(* IEC 61131-3 sources: ATCMcontrol_Engineering/src/TargetBase/Libs/ATCM_File, 19 files *)

(* ---- F_ERROR_STRING.st ---- *)
(*[[
    UserURL= "ATCMfile:F_ERROR_STRING.htm"
]]*)

(* F_ERROR_STRING
 * ----------------------------------------------------------------------------
 * Retrieves the error text that corresponds to the error number.
 *
 * in   ERRCD       Error code
 * out
 * ret              Error string
 *)
FUNCTION F_ERROR_STRING : STRING

VAR_INPUT
    ERRCD : DINT;
END_VAR

inline {STDLIB(f_error_string)}

END_FUNCTION

(* ---- F_FLUSH.st ---- *)
(*[[
    UserURL= "ATCMfile:F_FLUSH.htm"
]]*)

(* F_FLUSH
 * ----------------------------------------------------------------------------
 * This function causes any buffered output on all open files to be flushed.
 *
 * ret              Error code
 *)
FUNCTION F_FLUSH : DINT

inline {STDLIB(f_flush)}

END_FUNCTION

(* ---- F_GET_DISKFREESPACE.st ---- *)
(*[[
    UserURL= "ATCMfile:F_GET_DISKFREESPACE.htm"
]]*)

(* F_GET_DISKFREESPACE
 * ----------------------------------------------------------------------------
 * Retrieves the free disk space in kilo bytes for specified path.
 *
 * in   PATH        Path to the disk.
 * out  FREE_KB     Free disk space in kilo bytes.
 * ret              Error code
 *)
FUNCTION F_GET_DISKFREESPACE  : DINT

VAR_INPUT
    PATH : STRING;
END_VAR

VAR_OUTPUT
    FREE_KB : DINT;
END_VAR

inline {STDLIB(f_get_diskFreeSpace)}

END_FUNCTION

(* ---- F_SYNC_ARRAYREADFILE.st ---- *)
(*[[
    UserURL= "ATCMfile:F_SYNC_ARRAYREADFILE.htm"
]]*)

(* F_SYNC_ARRAYREADFILE
 * ----------------------------------------------------------------------------
 * Reads data from a file into an byte array.
 *
 * in   POS         Position in array where to store data.
 *                  (It is relative to lower bound (0 <= pos <= (hbound - lowbound).)
 * io   FILE        File instance to operate on.
 * io   LENGTH      in: bytes to read   out: bytes read
 * out  DATA        Data.
 * ret              Error flag: FALSE if successful - TRUE if failed.
 *)
FUNCTION F_SYNC_ARRAYREADFILE : BOOL
VAR_INPUT
    POS         : DINT;
END_VAR
VAR_IN_OUT
    FILE        : F_SYNC_FILE;
    LENGTH      : DINT;
END_VAR
VAR_OUTPUT
    DATA        : ARRAY OF BYTE;
END_VAR

inline {STDLIB(f_sync_arrayReadFile)}

END_FUNCTION

(* ---- F_SYNC_ARRAYWRITEFILE.st ---- *)
(*[[
    UserURL= "ATCMfile:F_SYNC_ARRAYWRITEFILE.htm"
]]*)

(* F_SYNC_ARRAYWRITEFILE
 * ----------------------------------------------------------------------------
 * Writes data from the given array to the specified file.
 *
 * in   DATA        Data to be written.
 * in   POS         Position in array where to store data.
 *                  (It is relative to lower bound (0 <= pos <= (hbound - lowbound).)
 * in   LENGTH      Bytes to be written.
 * io   FILE        File instance to operate on.
 * ret              Error flag: FALSE if successful - TRUE if failed.
 *)
FUNCTION F_SYNC_ARRAYWRITEFILE : BOOL

VAR_INPUT
    DATA        : ARRAY OF BYTE;
    POS         : DINT;
    LENGTH      : DINT;
END_VAR

VAR_IN_OUT
    FILE        : F_SYNC_FILE;
END_VAR

inline {STDLIB(f_sync_arrayWriteFile)}

END_FUNCTION

(* ---- F_SYNC_CLOSEFILE.st ---- *)
(*[[
    UserURL= "ATCMfile:F_SYNC_CLOSEFILE.htm"
]]*)

(* F_SYNC_CLOSEFILE
 * ----------------------------------------------------------------------------
 * Close the given file instance.
 *
 * io   FILE        File instance to operate on.
 * ret              Error flag: FALSE if successful - TRUE if failed.
 *)
FUNCTION F_SYNC_CLOSEFILE : BOOL

VAR_IN_OUT
    FILE        : F_SYNC_FILE;
END_VAR

inline {STDLIB(f_sync_closeFile)}

END_FUNCTION

(* ---- F_SYNC_COPYFILE.st ---- *)
(*[[
    UserURL= "ATCMfile:F_SYNC_COPYFILE.htm"
]]*)

(* F_SYNC_COPYFILE
 * ----------------------------------------------------------------------------
 * Copies file from source pathname to destination pathname.
 *
 * in   SrcPathName        Source pathname
 * in   DestPathName       Destination pathname
 *)
FUNCTION F_SYNC_COPYFILE : DINT

VAR_INPUT
SrcPathName  :   STRING;
DestPathName :   STRING;
END_VAR

inline {STDLIB(f_sync_copyFile)}

END_FUNCTION

(* ---- F_SYNC_CREATEDIRECTORY.st ---- *)
(*[[
    UserURL= "ATCMfile:F_SYNC_CREATEDIRECTORY.htm"
]]*)

(* F_SYNC_CREATEDIRECTORY
 * ----------------------------------------------------------------------------
 * Creates a new directory.
 *
 * io   FILE        File instance to operate on.
 * ret              Error flag: FALSE if successful - TRUE if failed.
 *)
FUNCTION F_SYNC_CREATEDIRECTORY : BOOL

VAR_IN_OUT
    FILE        : F_SYNC_FILE;
END_VAR

inline {STDLIB(f_sync_createDirectory)}

END_FUNCTION

(* ---- F_SYNC_DELETEFILE.st ---- *)
(*[[
    UserURL= "ATCMfile:F_SYNC_DELETEFILE.htm"
]]*)

(* F_SYNC_DELETEFILE
 * ----------------------------------------------------------------------------
 * Deletes the specified file.
 *
 * io   FILE        File instance to operate on.
 * ret              Error flag: FALSE if successful - TRUE if failed.
 *)
FUNCTION F_SYNC_DELETEFILE : BOOL

VAR_IN_OUT
    FILE        : F_SYNC_FILE;
END_VAR

inline {STDLIB(f_sync_deleteFile)}

END_FUNCTION

(* ---- F_SYNC_EXISTSFILE.st ---- *)
(*[[
    UserURL= "ATCMfile:F_SYNC_EXISTSFILE.htm"
]]*)

(* F_SYNC_EXISTSFILE
 * ----------------------------------------------------------------------------
 * Tests if the given file exists.
 *
 * io   FILE        File instance to operate on.
 * ret              Error flag: FALSE if successful - TRUE if failed.
 *)
FUNCTION F_SYNC_EXISTSFILE : BOOL

VAR_IN_OUT
    FILE        : F_SYNC_FILE;
END_VAR

inline {STDLIB(f_sync_existsFile)}

END_FUNCTION

(* ---- F_SYNC_GETSIZE.st ---- *)
(*[[
    UserURL= "ATCMfile:F_SYNC_GETSIZE.htm"
]]*)

(* F_SYNC_GETSIZE
 * ----------------------------------------------------------------------------
 * Gets the size of the given file.
 *
 * io   FILE        File instance to operate on.
 * out  SIZE        File size of given file.
 * ret              Error flag: FALSE if successful - TRUE if failed.
 *)
FUNCTION F_SYNC_GETSIZE : BOOL

VAR_IN_OUT
    FILE        : F_SYNC_FILE;
END_VAR

VAR_OUTPUT
    SIZE        : DINT;
END_VAR

inline {STDLIB(f_sync_getSize)}

END_FUNCTION

(* ---- F_SYNC_OPENFILE.st ---- *)
(*[[
    UserURL= "ATCMfile:F_SYNC_OPENFILE.htm"
]]*)

(* F_SYNC_OPENFILE
 * ----------------------------------------------------------------------------
 * Opens the given file.
 *
 * io   FILE        File instance to operate on.
 * ret              Error flag: FALSE if successful - TRUE if failed.
 *)
FUNCTION F_SYNC_OPENFILE : BOOL

VAR_IN_OUT
    FILE        : F_SYNC_FILE;
END_VAR

inline {STDLIB(f_sync_openFile)}

END_FUNCTION

(* ---- F_SYNC_READCSVFILE.st ---- *)
(*[[
    UserURL= "ATCMfile:F_SYNC_READCSVFILE.htm"
]]*)

(* F_SYNC_READCSVFILE
 * ----------------------------------------------------------------------------
 * Reads a record data from CSV file.
 *
 * in   FIELDSTRUCT specifies the maximum record field number and record field
 *                  format for all file records.
 * io   FILE        File instance to operate on.
 * out  DATA        Data.
 * ret              Error flag: FALSE if successful - TRUE if failed.
 *)
FUNCTION F_SYNC_READCSVFILE: BOOL

VAR_IN_OUT
    FILE        : F_SYNC_FILE;
END_VAR

VAR_INPUT
    FIELDSTRUCT : ARRAY OF BYTE;
    ACTRECORD   : DINT;
END_VAR

VAR_OUTPUT
    DATA        : ARRAY OF BYTE;
END_VAR

inline {STDLIB(f_sync_readCsvFile)}

END_FUNCTION

(* ---- F_SYNC_READFILE.st ---- *)
(*[[
    UserURL= "ATCMfile:F_SYNC_READFILE.htm"
]]*)

(* F_SYNC_READFILE
 * ----------------------------------------------------------------------------
 * Reads data from a file into a string.
 *
 * io   FILE        File instance to operate on.
 * io   LENGTH      in: bytes to read   out: bytes read
 * out  DATA        Data.
 * ret              Error flag: FALSE if successful - TRUE if failed.
 *)
FUNCTION F_SYNC_READFILE : BOOL
VAR_IN_OUT
    FILE        : F_SYNC_FILE;
    LENGTH      : DINT;
END_VAR
VAR_OUTPUT
    DATA        : STRING;
END_VAR

inline {STDLIB(f_sync_readFile)}

END_FUNCTION

(* ---- F_SYNC_READLINE.st ---- *)
(*[[
    UserURL= "ATCMfile:F_SYNC_READLINE.htm"
]]*)

(* F_SYNC_READLINE
 * ----------------------------------------------------------------------------
 * Reads a line from a file into a string.
 *
 * io   FILE        File instance to operate on.
 * out  DATA        Data.
 * ret              Error flag: FALSE if successful - TRUE if failed.
 *)
FUNCTION F_SYNC_READLINE : BOOL
VAR_IN_OUT
    FILE        : F_SYNC_FILE;
END_VAR
VAR_OUTPUT
    DATA        : STRING;
END_VAR

INLINE { STDLIB(f_sync_readLine) }

END_FUNCTION

(* ---- F_SYNC_RENAMEFILE.st ---- *)
(*[[
    UserURL= "ATCMfile:F_SYNC_RENAMEFILE.htm"
]]*)

(* F_SYNC_RENAMEFILE
 * ----------------------------------------------------------------------------
 * Renames the given file.
 *
 * in   NEWNAME     New file name.
 * io   FILE        File instance to operate on.
 * ret              Error flag: FALSE if successful - TRUE if failed.
 *)
FUNCTION F_SYNC_RENAMEFILE : BOOL

VAR_INPUT
    NEWNAME     : STRING;
END_VAR

VAR_IN_OUT
    FILE        : F_SYNC_FILE;
END_VAR

inline {STDLIB(f_sync_renameFile)}

END_FUNCTION

(* ---- F_SYNC_WRITECSVFILE.st ---- *)
(*[[
    UserURL= "ATCMfile:F_SYNC_WRITECSVFILE.htm"
]]*)

(* F_SYNC_READCSVFILE
 * ----------------------------------------------------------------------------
 * Writes a record data buffer to CSV file
 *
 * in   FIELDSTRUCT Maximum record field number and record field
 *                  format for all file records.
 * in   DATA        Data to be written.
 * io   FILE        File instance to operate on.
 * ret              Error flag: FALSE if successful - TRUE if failed.
 *)
FUNCTION F_SYNC_WRITECSVFILE: BOOL

VAR_IN_OUT
    FILE        : F_SYNC_FILE;
END_VAR

VAR_INPUT
    FIELDSTRUCT : ARRAY OF BYTE;
    ACTRECORD   : DINT;
    DATA        : ARRAY OF BYTE;
END_VAR

inline {STDLIB(f_sync_writeCsvFile)}

END_FUNCTION

(* ---- F_SYNC_WRITEFILE.st ---- *)
(*[[
    UserURL= "ATCMfile:F_SYNC_WRITEFILE.htm"
]]*)

(* F_SYNC_WRITEFILE
 * ----------------------------------------------------------------------------
 * Writes data from the given string to the specified file.
 *
 * in   DATA        Data to be written.
 * io   FILE        File instance to operate on.
 * ret              Error flag: FALSE if successful - TRUE if failed.
 *)
FUNCTION F_SYNC_WRITEFILE : BOOL
VAR_INPUT
    DATA        : STRING;
END_VAR
VAR_IN_OUT
    FILE        : F_SYNC_FILE;
END_VAR

inline {STDLIB(f_sync_writeFile)}

END_FUNCTION

(* ---- F_SYNC_WRITELINE.st ---- *)
(*[[
    UserURL= "ATCMfile:F_SYNC_WRITELINE.htm"
]]*)

(* F_SYNC_WRITELINE
 * ----------------------------------------------------------------------------
 * Writes a line to a file from a string.
 *
 * in   DATA        Data to be written.
 * io   FILE        File instance to operate on.
 * ret              Error flag: FALSE if successful - TRUE if failed.
 *)
FUNCTION F_SYNC_WRITELINE : BOOL
VAR_INPUT
    DATA        : STRING;
END_VAR
VAR_IN_OUT
    FILE        : F_SYNC_FILE;
END_VAR

INLINE { STDLIB(f_sync_writeLine) }

END_FUNCTION
